// TIA Portal V19 export
DATA_BLOCK "HmiInterface"   // DB114
// stored: Access Published, MemoryReserve 100, Namespace Unit2.Em6
   VAR
      em : "LAF_typeEmInterface";
      jobs : "LAF_typeJobsInterface";
      sequence : "LAF_typeSequenceInterface";
      cm1Vfd207 : "LEXCHANGETRAY_typeRollerVfdInterface";
      cm2SingalTM : "LEXCHANGETRAY_typeRollerIoSignalInterface_B2";
      em6Parameters : "LAF_typePlasticRollerEm6ParametersInterface";
   END_VAR
BEGIN
END_DATA_BLOCK
